FUNCTION F_degToRad : LREAL
VAR_INPUT
	fDeg : LREAL;
END_VAR
VAR
	piii :LREAL := 3.14;
END_VAR

F_degToRad := fDeg*(piii/180);

END_FUNCTION

(* stored: Version 1.1.0.1, ProductVersion 3.1.4024.10
   POU F_degToRad: Id {340d578b-4897-493a-ae17-8ad4ed18a680}, SpecialFunc None *)
